FUNCTION_BLOCK MOD_StateManager (* Module state manager: OPC UA methods Reset/Start/Stop/Abort/Clear(Session) answer [Accepted, ErrorID]; publishes the PackML State over OPC UA and on the module's state channel; RUN_RESETTING and RUN_STOPPING start the procedures, which answer with *_DONE or *_FAILED *)
  (* Standard: 61499-2 *)
  (* Version 0.1, 2026-09-28, Project contributors, AAU Smart Production Lab *)
  PACKAGE modlib;
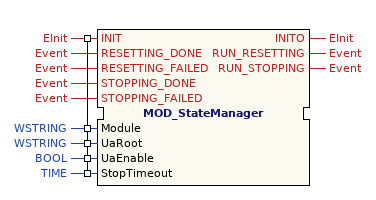
  EVENT_INPUT
    INIT : EInit WITH Module, UaRoot, UaEnable, StopTimeout;
    RESETTING_DONE;
    RESETTING_FAILED;
    STOPPING_DONE;
    STOPPING_FAILED;
  END_EVENT
  EVENT_OUTPUT
    INITO : EInit;
    RUN_RESETTING;
    RUN_STOPPING;
  END_EVENT
  VAR_INPUT
    Module : WSTRING;
    UaRoot : WSTRING;
    UaEnable : BOOL;
    StopTimeout : TIME := T#10s;
  END_VAR
  FBS
    Ids : modlib::MOD_StateIds;
    Owner : modlib::MOD_OwnerView;
    Reset : iec61499::net::SERVER_2_1;
    Start : iec61499::net::SERVER_2_1;
    Stop : iec61499::net::SERVER_2_1;
    Abort : iec61499::net::SERVER_2_1;
    Clear : iec61499::net::SERVER_2_1;
    Logic : modlib::MOD_StateLogic;
    PubUa : iec61499::net::PUBLISH_1;
    PubState : iec61499::net::PUBLISH_1(QI := TRUE);
    SubQuery : iec61499::net::SUBSCRIBE_0(QI := TRUE);
    SubAct : iec61499::net::SUBSCRIBE_1(QI := TRUE);
    Count : modlib::MOD_ActivityCount;
    Wd : iec61499::events::E_DELAY;
  END_FBS
  EVENT_CONNECTIONS
    INIT TO Ids.INIT;
    Ids.INITO TO Owner.INIT;
    Owner.INITO TO Reset.INIT;
    Reset.INITO TO Start.INIT;
    Start.INITO TO Stop.INIT;
    Stop.INITO TO Abort.INIT;
    Abort.INITO TO Clear.INIT;
    Clear.INITO TO PubUa.INIT;
    PubUa.INITO TO PubState.INIT;
    PubState.INITO TO SubQuery.INIT;
    SubQuery.INITO TO SubAct.INIT;
    SubAct.INITO TO PubUa.REQ;
    SubAct.INITO TO PubState.REQ;
    SubAct.INITO TO INITO;
    Owner.CHG TO Logic.OWNER_CHG;
    Reset.IND TO Logic.CMD_RESET;
    Logic.RSP_RESET TO Reset.RSP;
    Start.IND TO Logic.CMD_START;
    Logic.RSP_START TO Start.RSP;
    Stop.IND TO Logic.CMD_STOP;
    Logic.RSP_STOP TO Stop.RSP;
    Abort.IND TO Logic.CMD_ABORT;
    Logic.RSP_ABORT TO Abort.RSP;
    Clear.IND TO Logic.CMD_CLEAR;
    Logic.RSP_CLEAR TO Clear.RSP;
    Logic.CNF TO PubUa.REQ;
    Logic.CNF TO PubState.REQ;
    SubQuery.IND TO PubState.REQ;
    SubAct.IND TO Count.ACT;
    Count.CHG TO Logic.ACT;
    Logic.WD_START TO Wd.START;
    Logic.WD_STOP TO Wd.STOP;
    Wd.EO TO Logic.STOP_TIMEOUT;
    Logic.RUN_RESETTING TO RUN_RESETTING;
    Logic.RUN_STOPPING TO RUN_STOPPING;
    RESETTING_DONE TO Logic.RESETTING_DONE;
    RESETTING_FAILED TO Logic.RESETTING_FAILED;
    STOPPING_DONE TO Logic.STOPPING_DONE;
    STOPPING_FAILED TO Logic.STOPPING_FAILED;
  END_CONNECTIONS
  DATA_CONNECTIONS
    Module TO Ids.Module;
    Module TO Owner.Module;
    UaRoot TO Ids.UaRoot;
    UaEnable TO Reset.QI;
    UaEnable TO Start.QI;
    UaEnable TO Stop.QI;
    UaEnable TO Abort.QI;
    UaEnable TO Clear.QI;
    UaEnable TO PubUa.QI;
    StopTimeout TO Wd.DT;
    Owner.Owner TO Logic.Owner;
    Ids.IdReset TO Reset.ID;
    Reset.RD_1 TO Logic.S_Reset;
    Logic.Accepted TO Reset.SD_1;
    Logic.ErrorID TO Reset.SD_2;
    Ids.IdStart TO Start.ID;
    Start.RD_1 TO Logic.S_Start;
    Logic.Accepted TO Start.SD_1;
    Logic.ErrorID TO Start.SD_2;
    Ids.IdStop TO Stop.ID;
    Stop.RD_1 TO Logic.S_Stop;
    Logic.Accepted TO Stop.SD_1;
    Logic.ErrorID TO Stop.SD_2;
    Ids.IdAbort TO Abort.ID;
    Abort.RD_1 TO Logic.S_Abort;
    Logic.Accepted TO Abort.SD_1;
    Logic.ErrorID TO Abort.SD_2;
    Ids.IdClear TO Clear.ID;
    Clear.RD_1 TO Logic.S_Clear;
    Logic.Accepted TO Clear.SD_1;
    Logic.ErrorID TO Clear.SD_2;
    Ids.IdPub TO PubUa.ID;
    Ids.IdState TO PubState.ID;
    Ids.IdQuery TO SubQuery.ID;
    Ids.IdAct TO SubAct.ID;
    Logic.State TO PubUa.SD_1;
    Logic.State TO PubState.SD_1;
    SubAct.RD_1 TO Count.Delta;
    Count.AllIdle TO Logic.AllIdle;
  END_CONNECTIONS
END_FUNCTION_BLOCK
